// TIA Portal V20 export
DATA_BLOCK "ComSd"   // DB362
{ S7_Optimized_Access := 'FALSE' }
// stored: AutoNumber false
   VAR
      Plc : "TypeHeaderPlc";   // Header Plc
      Pc : "TypeHeaderPcGld";   // Header Pc
      Data : Struct
         config : Struct   // config
            "Version" : Int;   // version info
            spare2 : Int;
            spare3 : Int;
            spare4 : Int;
         END_STRUCT;
         control : Struct   // control
            spare : Bool;
         END_STRUCT;
         safety : Struct   // safety
            AreaLaserOn : Bool;   // area laser on
            AreaAdjustmentOn : Bool;   // area adjustment on
            AreaXrayOn : Bool;   // area X-Ray on
            spare : Bool;
         END_STRUCT;
         status : Struct   // status
            ready : Bool;   // plc ready
            err : Bool;   // plc error
         END_STRUCT;
         Scanner : "TypeAxisSd";   // adjustment scanner
         Top : "TypeAxisSd";   // adjustment top
         Left : "TypeAxisSd";   // adjustment left
         Right : "TypeAxisSd";   // adjustment right
         Measure : Struct   // measuring sensor for random width/thickness
            ActValueTop : DInt;   // actual value [mm/10]
            ActValueLeft : DInt;   // actual value [mm/10]
            ActValueRight : DInt;   // actual value [mm/10]
            Thickness : DInt;   // thickness [mm/10]
            Width : DInt;   // width [mm/10]
            SetCalibratePosTopOk : Bool;   // set calibrated position for sensor top ok
            SetCalibratePosLeftOk : Bool;   // set calibrated position for sensor left ok
            SetCalibratePosRightOk : Bool;   // set calibrated position for sensor right ok
         END_STRUCT;
         PlcInputNormal : Struct   // plc Input normal
            "I0.0" : Bool;
            "I0.1" : Bool;
            "I0.2" : Bool;
            "I0.3" : Bool;
            "I0.4" : Bool;
            "I0.5" : Bool;
            "I0.6" : Bool;
            "I0.7" : Bool;
            "I1.0" : Bool;
            "I1.1" : Bool;
            "I1.2" : Bool;
            "I1.3" : Bool;
            "I1.4" : Bool;
            "I1.5" : Bool;
            "I1.6" : Bool;
            "I1.7" : Bool;
            "I2.0" : Bool;
            "I2.1" : Bool;
            "I2.2" : Bool;
            "I2.3" : Bool;
            "I2.4" : Bool;
            "I2.5" : Bool;
            "I2.6" : Bool;
            "I2.7" : Bool;
         END_STRUCT;
         PlcInputSafety : Struct   // plc Input safety
            "I800.0" : Bool;
            "I800.1" : Bool;
            "I800.2" : Bool;
            "I800.3" : Bool;
            "I808.0" : Bool;
            "I808.1" : Bool;
            "I808.2" : Bool;
            "I808.3" : Bool;
            "I816.0" : Bool;
            "I816.1" : Bool;
            "I816.2" : Bool;
            "I816.3" : Bool;
            "I824.0" : Bool;
            "I824.1" : Bool;
            "I824.2" : Bool;
            "I824.3" : Bool;
         END_STRUCT;
         PlcOutputNormal : Struct   // plc output normal
            "Q0.0" : Bool;
            "Q0.1" : Bool;
            "Q0.2" : Bool;
            "Q0.3" : Bool;
            "Q0.4" : Bool;
            "Q0.5" : Bool;
            "Q0.6" : Bool;
            "Q0.7" : Bool;
            "Q1.0" : Bool;
            "Q1.1" : Bool;
            "Q1.2" : Bool;
            "Q1.3" : Bool;
            "Q1.4" : Bool;
            "Q1.5" : Bool;
            "Q1.6" : Bool;
            "Q1.7" : Bool;
            "Q2.0" : Bool;
            "Q2.1" : Bool;
            "Q2.2" : Bool;
            "Q2.3" : Bool;
            "Q2.4" : Bool;
            "Q2.5" : Bool;
            "Q2.6" : Bool;
            "Q2.7" : Bool;
         END_STRUCT;
         PlcOutputSafety : Struct   // plc output safety
            "Q900.0" : Bool;
            "Q900.1" : Bool;
            "Q900.2" : Bool;
            "Q900.3" : Bool;
            "Q908.0" : Bool;
            "Q908.1" : Bool;
            "Q908.2" : Bool;
            "Q908.3" : Bool;
         END_STRUCT;
         res : Array[1..200] of Byte;
      END_STRUCT;
   END_VAR
BEGIN
END_DATA_BLOCK
